FUNCTION_BLOCK UDIntPointerComparer EXTENDS Object IMPLEMENTS IPointerComparer
VAR
	_ClassName : STRING := __POUNAME();
END_VAR

{attribute 'monitoring' := 'call'}
PROPERTY ClassName : STRING
GET
ClassName := _ClassName;
END_GET
END_PROPERTY

{attribute "object_name" := "Compare"}
METHOD Compare : COMPARISION_RESULT
VAR_INPUT
	left : PVOID;
	right : PVOID;
END_VAR
VAR
	leftPointer : POINTER TO UDINT; 
	rightPointer : POINTER TO UDINT; 
END_VAR
IF left = 0 AND right = 0 THEN
	Compare := COMPARISION_RESULT.FIRST_EQUAL_TO_SECOND;
	RETURN;
END_IF

IF left = 0 THEN
	Compare := COMPARISION_RESULT.FIRST_LESS_THAN_SECOND;
	RETURN;	
END_IF

IF right = 0 THEN
	Compare := COMPARISION_RESULT.FIRST_GREATER_THAN_SECOND;
	RETURN;	
END_IF

leftPointer := left;
rightPointer := right;

IF leftPointer^ < rightPointer^ THEN
	Compare := COMPARISION_RESULT.FIRST_LESS_THAN_SECOND;
ELSIF leftPointer^ > rightPointer^ THEN
	Compare := COMPARISION_RESULT.FIRST_GREATER_THAN_SECOND;
ELSE
	Compare := COMPARISION_RESULT.FIRST_EQUAL_TO_SECOND;	
END_IF
END_METHOD

{attribute 'monitoring' := 'call'}
PROPERTY Size : ULINT
GET
Size := XSIZEOF(THIS^);
END_GET
END_PROPERTY

END_FUNCTION_BLOCK

(* stored: Version 1.1.0.1
   POU UDIntPointerComparer: Id {9fdbb449-9d2c-44b0-b6e5-69ef7ba3e1c9}, SpecialFunc None
   Property ClassName: Id {59b4cb09-ce27-4cf2-822b-22a02ff2a32e}
   Get Get: Id {773aab9c-6554-4fb1-b71d-4aea6762494a}
   Method Compare: Id {6842a060-1190-4443-a2cb-0127a057a5a4}
   Property Size: Id {a227353e-8503-4785-9150-98b9fd2830da}
   Get Get: Id {697e7265-e590-4caa-9214-5a5ab64fe284} *)
